(* IEC 61131-3 sources: SMARTT/OT_Emulation_Data_Broker/PLCs/RX_PowerCtrl/build, 2 files *)

(* ---- plc.st ---- *)
TYPE
  LOGLEVEL : (CRITICAL, WARNING, INFO, DEBUG) := INFO;
END_TYPE

FUNCTION_BLOCK LOGGER
  VAR_INPUT
    TRIG : BOOL;
    MSG : STRING;
    LEVEL : LOGLEVEL := INFO;
  END_VAR
  VAR
    TRIG0 : BOOL;
  END_VAR

  IF TRIG AND NOT TRIG0 THEN
  {{
   LogMessage(GetFbVar(LEVEL),(char*)GetFbVar(MSG, .body),GetFbVar(MSG, .len));
  }}
  END_IF;
  TRIG0:=TRIG;
END_FUNCTION_BLOCK

FUNCTION_BLOCK python_eval
  VAR_INPUT
    TRIG : BOOL;
    CODE : STRING;
  END_VAR
  VAR_OUTPUT
    ACK : BOOL;
    RESULT : STRING;
  END_VAR
  VAR
    STATE : DWORD;
    BUFFER : STRING;
    PREBUFFER : STRING;
    TRIGM1 : BOOL;
    TRIGGED : BOOL;
  END_VAR

  {extern void __PythonEvalFB(int, PYTHON_EVAL*);__PythonEvalFB(0, data__);}
END_FUNCTION_BLOCK

FUNCTION_BLOCK python_poll
  VAR_INPUT
    TRIG : BOOL;
    CODE : STRING;
  END_VAR
  VAR_OUTPUT
    ACK : BOOL;
    RESULT : STRING;
  END_VAR
  VAR
    STATE : DWORD;
    BUFFER : STRING;
    PREBUFFER : STRING;
    TRIGM1 : BOOL;
    TRIGGED : BOOL;
  END_VAR

  {extern void __PythonEvalFB(int, PYTHON_EVAL*);__PythonEvalFB(1,(PYTHON_EVAL*)(void*)data__);}
END_FUNCTION_BLOCK

FUNCTION_BLOCK python_gear
  VAR_INPUT
    N : UINT;
    TRIG : BOOL;
    CODE : STRING;
  END_VAR
  VAR_OUTPUT
    ACK : BOOL;
    RESULT : STRING;
  END_VAR
  VAR
    py_eval : python_eval;
    COUNTER : UINT;
    ADD10_OUT : UINT;
    EQ13_OUT : BOOL;
    SEL15_OUT : UINT;
    AND7_OUT : BOOL;
  END_VAR

  ADD10_OUT := ADD(COUNTER, 1);
  EQ13_OUT := EQ(N, ADD10_OUT);
  SEL15_OUT := SEL(EQ13_OUT, ADD10_OUT, 0);
  COUNTER := SEL15_OUT;
  AND7_OUT := AND(EQ13_OUT, TRIG);
  py_eval(TRIG := AND7_OUT, CODE := CODE);
  ACK := py_eval.ACK;
  RESULT := py_eval.RESULT;
END_FUNCTION_BLOCK

PROGRAM RX_PowerCTRL
  VAR
    TIME_IN : REAL;
    TIME_OUT : REAL;
    RX_Power : REAL;
    CTRL_RXPowerSetpoint : REAL := 0.0;
    MANIPIO_CONTROL : REAL := 0.0;
    KPI : REAL := -100.0;
    Ti : REAL := 60.0;
    SET_POINT : REAL := 1.0;
    INIT : REAL := 90.0;
    TIME_COMP : REAL := 150.0;
  END_VAR

  TIME_OUT := TIME_IN;

  IF TIME_OUT >= TIME_COMP THEN
    TIME_COMP := TIME_OUT + 150.0;
    CTRL_RXPowerSetpoint := CTRL_RXPowerSetpoint + 0.1;
  END_IF;
END_PROGRAM

CONFIGURATION Config0

  RESOURCE Res0 ON PLC
    TASK task0(INTERVAL := T#100ms,PRIORITY := 0);
    PROGRAM instance0 WITH task0 : RX_PowerCTRL;
  END_RESOURCE
END_CONFIGURATION

(* ---- generated_plc.st ---- *)
PROGRAM RX_PowerCTRL
  VAR
    TIME_IN AT %MD0 : REAL;
    TIME_OUT AT %MD1 : REAL;
    RX_Power AT %MD2 : REAL;
    CTRL_RXPowerSetpoint AT %MD3 : REAL := 0.0;
    MANIPIO_CONTROL AT %MD4 : REAL := 0.0;
    KPI AT %MD5 : REAL := -100.0;
    Ti AT %MD6 : REAL := 60.0;
    SET_POINT AT %MD7 : REAL := 1.0;
    INIT AT %MD8 : REAL := 90.0;
    TIME_COMP AT %MD9 : REAL := 150.0;
  END_VAR

  TIME_OUT := TIME_IN;

  IF TIME_OUT >= TIME_COMP THEN
    TIME_COMP := TIME_OUT + 150.0;
    CTRL_RXPowerSetpoint := CTRL_RXPowerSetpoint + 0.1;
  END_IF;
END_PROGRAM

CONFIGURATION Config0

  RESOURCE Res0 ON PLC
    TASK task0(INTERVAL := T#100ms,PRIORITY := 0);
    PROGRAM instance0 WITH task0 : RX_PowerCTRL;
  END_RESOURCE
END_CONFIGURATION
